TYPE hmiCommands_TypeStruct :
STRUCT
	
	orderControl	: orderHmiCommands_TypeStruct;
	lineControl		: lineControlHmiCommands_TypeStruct;	
	slitter1		: slitterCommands_TypeStruct;
	upperKnife		: rotaryKnifeCommands_TypeStruct;
	lowerKnife		: rotaryKnifeCommands_TypeStruct;	
	
	lowerStacker	: hmiCommandsSimpleStacker_TypeStruct;
	upperStacker	: hmiCommandsComplexStacker_TypeStruct;
	
END_STRUCT
END_TYPE

(* stored: Version 1.1.0.1
   DUT hmiCommands_TypeStruct: Id {e9fcde45-7d62-44c1-a627-931f7dd406d1} *)
